// TIA Portal project "CELDA_CORTE_EQUIPO_DEPORTIVO" (V14)

(* hardware
DEVICE "S71500/ET200MP station_16"  S7-1500 station
   slot 0: "Perfil soporte_0"  Rack  6ES7 590-1***0-0AA0
   slot 1: "AUTO_CELDA_DE_CORTE"  CPU 1516F-3 PN/DP  6ES7 516-3FN00-0AB0  V1.8
      slot 3: "Display de la CPU_1"  6ES7591-1BA00-0AA0
   slot 2: "DI 32x24VDC BA_1"  DI 32x24VDC BA  6ES7 521-1BL10-0AA0  V1.0
   slot 3: "DQ 32x24VDC/0.5A BA_1"  DQ 32x24VDC/0.5A BA  6ES7 522-1BL10-0AA0  V1.0
   slot 4: "DI 32x24VDC BA_2"  DI 32x24VDC BA  6ES7 521-1BL10-0AA0  V1.0
*)

// ===== PLC "AUTO_CELDA_DE_CORTE"  CPU 1516F-3 PN/DP =====

VAR_GLOBAL   // PLC tag table "Tabla de variables estándar"
   ""ON"" AT %I0.0 : Bool;
   ""SC1"" AT %I1.3 : Bool;
   ""SC2"" AT %I1.4 : Bool;
   ""SC3_Izquierda"" AT %I1.5 : Bool;
   ""SL1"" AT %I1.6 : Bool;
   ""SL2"" AT %I1.7 : Bool;
   ""SL3_Izquierda"" AT %I2.0 : Bool;
   ""SS1"" AT %I2.1 : Bool;
   ""SS2"" AT %I2.2 : Bool;
   ""SS3_Izquierda"" AT %I2.3 : Bool;
   ""OFF"" AT %I0.1 : Bool;
   ""MA"" AT %I2.5 : Bool;
   ""MB"" AT %I2.6 : Bool;
   ""señal_pirómetro"" AT %IW6 : Word;
   ""FC1_C"" AT %I0.2 : Bool;
   ""FC1_E"" AT %I0.3 : Bool;
   ""FC2_C"" AT %I0.4 : Bool;
   ""FC2_E"" AT %I0.5 : Bool;
   ""FC3_C"" AT %I0.6 : Bool;
   ""FC3_E"" AT %I0.7 : Bool;
   ""pieza_válida_corte"" AT %I4.0 : Bool;
   ""pieza_válida_laminado"" AT %I4.1 : Bool;
   ""pieza_válida_serigrafía"" AT %I2.7 : Bool;
   ""SC3_Derecha"" AT %I3.0 : Bool;
   ""SL3_Derecha"" AT %I3.1 : Bool;
   ""SS3_Derecha"" AT %I2.4 : Bool;
   ""SB1_superior"" AT %I3.2 : Bool;
   ""SB1_inferior"" AT %I3.3 : Bool;
   ""SB2_superior"" AT %I3.4 : Bool;
   ""SB2_inferior"" AT %I3.5 : Bool;
   ""SC0"" AT %I3.6 : Bool;
   ""SL0"" AT %I3.7 : Bool;
   ""SS0"" AT %I4.2 : Bool;
   ""aviso_brazo1_en_posición"" AT %I4.3 : Bool;
   ""aviso_brazo2_en_posición"" AT %I4.4 : Bool;
   ""comando_alimentar_brazo1"" AT %I4.5 : Bool;
   ""comando_alimentar_brazo2"" AT %I4.6 : Bool;
   ""aviso_fin_de_maniobra_brazo1"" AT %I4.7 : Bool;
   ""aviso_fin_de_maniobra_brazo2"" AT %I5.1 : Bool;
   ""aviso_fin_tratamiento_corte"" AT %I5.2 : Bool;
   ""aviso_fin_tratamiento_laminado"" AT %I5.3 : Bool;
   ""aviso_fin_tratamiento_serigrafiado"" AT %I5.4 : Bool;
   ""aviso_máquina_corte_en_posición"" AT %I5.5 : Bool;
   ""aviso_máquina_laminado_en_posición"" AT %I5.6 : Bool;
   ""aviso_máquina_serigrafiado_en_posición"" AT %I5.7 : Bool;
   ""EMER"" AT %I1.1 : Bool;
   ""Rearme"" AT %I1.0 : Bool;
   ""LÁMPARA_IR"" AT %Q2.0 : Bool;
   ""EXP1"" AT %Q0.6 : Bool;
   ""COMP1"" AT %Q0.7 : Bool;
   ""EXP2"" AT %Q1.0 : Bool;
   ""COMP2"" AT %Q1.1 : Bool;
   ""EXP3"" AT %Q1.2 : Bool;
   ""COMP3"" AT %Q1.3 : Bool;
   ""ALIMENTAR_B1"" AT %Q0.3 : Bool;
   ""EXTRAER_SUPERIOR_B1"" AT %Q0.4 : Bool;
   ""EXTRAER_INFERIOR_B1"" AT %Q0.5 : Bool;
   ""ALIMENTAR_B2"" AT %Q0.0 : Bool;
   ""EXTRAER_SUPERIOR_B2"" AT %Q0.1 : Bool;
   ""EXTRAER_INFERIOR_B2"" AT %Q0.2 : Bool;
   ""CINTA_VOLCADO_Laminado"" AT %Q2.3 : Bool;
   ""CINTA_VOLCADO_Corte"" AT %Q2.2 : Bool;
   ""MÁQUINA_CORTE_ON"" AT %Q2.6 : Bool;
   ""MÁQUINA_LAMINADO_ON"" AT %Q2.5 : Bool;
   ""MÁQUINA_SERIGRAFIADO_ON"" AT %Q2.4 : Bool;
   ""CINTA_VOLCADO_Serigrafiado"" AT %Q2.1 : Bool;
   ""CINTA1_H"" AT %Q1.4 : Bool;
   ""CINTA1_A"" AT %Q1.5 : Bool;
   ""CINTA2_H"" AT %Q1.6 : Bool;
   ""CINTA2_A"" AT %Q1.7 : Bool;
END_VAR